FUNCTION_BLOCK FB_Base

END_FUNCTION_BLOCK

(* stored: Version 1.1.0.1
   POU FB_Base: Id {77777777-7777-7777-7777-777777777701} *)
